// TIA Portal V20 export
// export: Created 2025-12-01T14:56:12.1175121Z, ExportSetting None, DisplayName Totally Integrated Automation Portal, DisplayVersion V20 Update 3, DisplayName TIA Portal Openness, DisplayVersion V20 Update 3, DisplayName TIA Portal Version Control Interface, DisplayVersion V20 Update 3, DisplayName STEP 7 Professional, DisplayVersion V20 Update 3, DisplayName STEP 7 Safety, DisplayVersion V20 Update 2, DisplayName WinCC Basic/Comfort/Advanced, DisplayVersion V20 Update 3, DisplayName WinCC Professional, DisplayVersion V20 Update 3, DisplayName WinCC Unified, DisplayVersion V20 Update 3
TYPE "MoviManualMesa"
   STRUCT
      Avance_Rod : Bool;   // Pulsador MAN AVANCE RODILLOS
      Retroceso_Rod : Bool;   // Pulsador MAN RETROCEDE RODILLOS
      Avance_Cad : Bool;   // Pulsador MAN AVANCE CADENAS
      Retroceso_Cad : Bool;   // Pulsador MAN RETROCEDE CADENAS
      Elevacion : Bool;   // Pulsador MAN SUBIR TRANSFER /MAQUETA/MESA ELEVADORA
      Descenso : Bool;   // Pulsador MAN BAJAR TRANSFER /MAQUETA/MESA ELEVADORA
      Subir_TP1 : Bool;   // Pulsador MAN SUBIR TOPE 1
      Bajar_TP1 : Bool;   // Pulsador MAN BAJAR TOPE 1
      Giro_0 : Bool;   // Pulsador MAN GIRAR HACIA POSICION 0
      Giro_90 : Bool;   // Pulsador MAN GIRAR HACIA POSICION 90
      Giro_180 : Bool;   // Pulsador MAN GIRAR HACIA POSICION 180
      Subir_TP2 : Bool;   // Pulsador MAN SUBIR TOPE 2
      Bajar_TP2 : Bool;   // Pulsador MAN BAJAR TOPE 2
      Byte1_bit5 : Bool;   // …
      Byte1_bit6 : Bool;   // …
      Byte1_bit7 : Bool;   // ..
      SimulRod_AvSig : Bool;   // Mov SIMULTANEO AVANCE RODILLOS SIGUIENTE
      SimulRod_AvAnt : Bool;   // Mov SIMULTANEO AVANCE RODILLOS ANTERIOR
      SimulRod_RtSig : Bool;   // Mov SIMULTANEO RETROCEDE RODILLOS SIGUIENTE
      SimulRod_RtAnt : Bool;   // Mov SIMULTANEO RETROCEDE RODILLOS ANTERIOR
      Byte2_bit4 : Bool;   // …
      Byte2_bit5 : Bool;   // …
      Byte2_bit6 : Bool;   // …
      Byte2_bit7 : Bool;   // …
      SimulCad_AvSig : Bool;   // Mov SIMULTANEO AVANCE CADENAS SIGUIENTE
      SimulCad_AvAnt : Bool;   // Mov SIMULTANEO AVANCE CADENAS ANTERIOR
      SimulCad_RtSig : Bool;   // Mov SIMULTANEO RETROCEDE CADENAS SIGUIENTE
      SimulCad_RtAnt : Bool;   // Mov SIMULTANEO RETROCEDE CADENAS ANTERIOR
      Byte3_bit4 : Bool;   // ..
      Byte3_bit5 : Bool;   // …
      Byte3_bit6 : Bool;   // …
      Byte3_bit7 : Bool;   // …
      Byte4_bit0 : Bool;   // …
      Byte4_bit1 : Bool;   // …
      Byte4_bit2 : Bool;   // …
      Byte4_bit3 : Bool;   // …
      Byte4_bit4 : Bool;   // …
      Byte4_bit5 : Bool;   // …
      Byte4_bit6 : Bool;   // …
      Byte4_bit7 : Bool;   // …
      Byte5_bit0 : Bool;   // ...
      Byte5_bit1 : Bool;   // ...
      Reset_Mesa : Bool;   // ...
      Rearme : Bool;   // ...
      Byte5_bit4 : Bool;   // ...
      Byte5_bit5 : Bool;   // ...
      Byte5_bit6 : Bool;   // ...
      Byte5_bit7 : Bool;   // ...
      Byte6_bit0 : Bool;   // ...
      Byte6_bit1 : Bool;   // ...
      Byte6_bit2 : Bool;   // ...
      Byte6_bit3 : Bool;   // ...
      Byte6_bit4 : Bool;   // ...
      Byte6_bit5 : Bool;   // ...
      Byte6_bit6 : Bool;   // ...
      Byte6_bit7 : Bool;   // ...
      Byte7_bit0 : Bool;   // ...
      Byte7_bit1 : Bool;   // ...
      Byte7_bit2 : Bool;   // ...
      Byte7_bit3 : Bool;   // ...
      Byte7_bit4 : Bool;   // ...
      Byte7_bit5 : Bool;   // ...
      Byte7_bit6 : Bool;   // ...
      Byte7_bit7 : Bool;   // …
   END_STRUCT;
END_TYPE
